// TIA Portal V18 export
TYPE "MEStoPLC_MainCheckIn"
// stored: IsFailsafeCompliant false
   STRUCT
      "M-OrderNum" : String[48];   // 订单号
      "M-PartType" : String[28];   // MES上线工位专用，下发主工件型号MN
      "M-PartID" : String[48];   // MES上线工位专用，下发主工件序列号SN
      "M-PartIDReqDone" : Bool;   // MES响应PLC请求当前产品能否生产
      "M-RecipeDone" : Bool;   // MES响应PLC请求参数下发完成标志位，MES置位信号后，PLC立即复位请求下发信号P-ReqMes
      "M-PartOK" : Bool;   // 工件可加工标志位，PLC收到M-ReqMesDone+此信号后可开始加工
      "M-PartNG" : Bool;   // 工件可不加工标志位，PLC收到M-ReqMesDone+此信号后可放行
      "M-PartStatus" : Byte;   // 1=正常，2=返修，3=标定
      "M-PartRouting" : Byte;   // 转台路由指示工位专用状态字，0、1、2等含义来指定路线
      "M-RecipeVer" : String[18];   // 工艺参数版本号
      "M-ErrorCode" : Int;   // 【预留】“M-ErrorMsg”失效的时候启用
      "M-ErrorMsg" : String[98];   // P-ReqMes请求Mes标志位收到后，如果Mes对请求的数据校验有异常，写入相应中文字符串，M-ReqMesDone信号超时后将中文字符串显示到HMI
      Reserve : Array[1..744] of Byte;   // Main-CheckIN预留
   END_STRUCT;
END_TYPE
